FUNCTION_BLOCK FB_CylinderNexaHmi EXTENDS FB_Cylinder
VAR
	(* Hmi *)       			
	_Hmi						: TcNexa_Devices_TcDeviceBase.FB_DeviceNexaHmi(deviceType:= 'cylinders');
	_onHmiConnection			: Tc2_Standard.R_TRIG;
	_isHmiConnected				: BOOL;
	_commandNameHP				: STRING;
	_commandNameWP				: STRING;
	_manualMode					: BOOL;
	_onResponseError			: Tc2_Standard.R_TRIG;
	_onResponsePass				: Tc2_Standard.R_TRIG;
	_interlockHPforOtherDevices	: STRING;
	_interlockWPforOtherDevices	: STRING;
	(* Control VAR *)
	_lastNotUsedSensorHP		: BOOL;
	_lastSensorHP				: BOOL;
	_lastNotUsedSensorWP		: BOOL;
	_lastSensorWP				: BOOL;
	_message					: STRING(255);
	_lastMessage				: STRING(255);
	(* Buttons *)
	_ButtonHP					: TcNexa_Devices_TcDeviceBase.FB_DeviceButtonNexaHmi(
									Hmi			:= _Hmi, 
									topic		:= 'general/buttons/HP/');
	_ButtonWP					: TcNexa_Devices_TcDeviceBase.FB_DeviceButtonNexaHmi(
									Hmi			:= _Hmi, 
									topic		:= 'general/buttons/WP/');
	(* Commands *)
	_requestHP					: BOOL;
	_requestWP					: BOOL;
END_VAR

METHOD PROTECTED _handleButtons
VAR_INPUT
END_VAR
(*----------------------------------------------------------------------------------------------*)
_ButtonHP.enabled:= NOT _interlockHP AND _manualMode;
_ButtonHP.focused:= valveHP;
_ButtonHP.name:= _commandNameHP;
_ButtonHP.FB_main();
(*----------------------------------------------------------------------------------------------*)
_ButtonWP.enabled:= NOT _interlockWP AND _manualMode;
_ButtonWP.focused:= valveWP;
_ButtonWP.name:= _commandNameWP;
_ButtonWP.FB_main();
(*----------------------------------------------------------------------------------------------*)
IF NOT _manualMode THEN RETURN; END_IF
IF _ButtonHP.onTap THEN	_requestHP:= TRUE; END_IF
IF _ButtonWP.onTap THEN	_requestWP:= TRUE; END_IF
(*----------------------------------------------------------------------------------------------*)
END_METHOD

METHOD PROTECTED _handleManual
VAR_INPUT
END_VAR
IF NOT _manualMode THEN
	_requestHP:= FALSE;
	_requestWP:= FALSE;
	_message:= 'Movement blocked: Not in manual mode';
ELSIF _interlockHP AND NOT _inHP THEN
	_message:= Tc2_Standard.CONCAT(STR1:= _commandNameHP, ' blocked: ');
	_message:= Tc2_Standard.CONCAT(STR1:= _message, _interlockMessageHP);
ELSIF _interlockWP AND NOT _inWP THEN
	_message:= Tc2_Standard.CONCAT(STR1:= _commandNameWP, ' blocked: ');
	_message:= Tc2_Standard.CONCAT(STR1:= _message, _interlockMessageWP);
ELSE
	_message:= '';
	(* HP *)
	IF _requestHP THEN
		moveToHP(Response:= _InternalResponse);
		_requestHP:= FALSE;
	END_IF
	(* HP *)
	IF _requestWP THEN
		moveToWP(Response:= _InternalResponse);
		_requestWP:= FALSE;
	END_IF
END_IF
END_METHOD

METHOD PROTECTED _onConnection
VAR_INPUT
END_VAR
IF NOT _onHmiConnection.Q THEN RETURN; END_IF

(* Publish *)
_Hmi.publish(
	topic	:= 'general/sensorTagHP',
	payload	:= _sensorTagHP);
_Hmi.publish(
	topic	:= 'general/sensorTagWP',
	payload	:= _sensorTagWP);
END_METHOD

METHOD PROTECTED _publishTopics
VAR_INPUT
END_VAR
IF NOT _isHmiConnected THEN RETURN; END_IF
(*----------------------------------------------------------------------------------------------*)
IF (_lastNotUsedSensorHP <> _notUsedSensorHP) OR _onHmiConnection.Q THEN
	_lastNotUsedSensorHP:= _notUsedSensorHP;
	_Hmi.publish(
		topic	:= 'general/notUsedSensorHP',
		payload	:= BOOL_TO_STRING(_notUsedSensorHP));
END_IF
(*----------------------------------------------------------------------------------------------*)
IF (_lastSensorHP <> sensorHP) OR _onHmiConnection.Q THEN
	_lastSensorHP:= sensorHP;
	_Hmi.publish(
		topic	:= 'general/sensorHP',
		payload	:= BOOL_TO_STRING(sensorHP));
END_IF
(*----------------------------------------------------------------------------------------------*)
IF (_lastNotUsedSensorWP <> _notUsedSensorWP) OR _onHmiConnection.Q THEN
	_lastNotUsedSensorWP:= _notUsedSensorWP;
	_Hmi.publish(
		topic	:= 'general/notUsedSensorWP',
		payload	:= BOOL_TO_STRING(_notUsedSensorWP));
END_IF
(*----------------------------------------------------------------------------------------------*)
IF (_lastSensorWP <> sensorWP) OR _onHmiConnection.Q THEN
	_lastSensorWP:= sensorWP;
	_Hmi.publish(
		topic	:= 'general/sensorWP',
		payload	:= BOOL_TO_STRING(sensorWP));
END_IF
(*----------------------------------------------------------------------------------------------*)
IF (_message <> _lastMessage) OR _onHmiConnection.Q THEN
	_lastMessage:= _message;
	_Hmi.publish(
		topic	:= 'general/message',
		payload	:= _message);
END_IF
(*----------------------------------------------------------------------------------------------*)
END_METHOD

METHOD FB_init : BOOL
VAR_INPUT
	bInitRetains 	: BOOL; // if TRUE, the retain variables are initialized (warm start / cold start)
	bInCopyCode 	: BOOL;  // if TRUE, the instance afterwards gets moved into the copy code (online change)
	name			: STRING;
	tag				: STRING;
	sensorTagHP		: STRING;
	sensorTagWP		: STRING;
	commandNameHP	: STRING;
	commandNameWP	: STRING;
	cellTag			: STRING;
	stationTag		: STRING;
END_VAR
THIS^._commandNameHP:= commandNameHP;
THIS^._commandNameWP:= commandNameWP;

THIS^._Hmi.cellTag:= cellTag;
THIS^._Hmi.stationTag:= stationTag;
THIS^._Hmi.deviceTag:= tag;
THIS^._Hmi.deviceName:= name;

_interlockHPforOtherDevices:= Tc2_Standard.CONCAT(STR1:= _nameTag, STR2:= ' not in ');
_interlockHPforOtherDevices:= Tc2_Standard.CONCAT(STR1:= _interlockHPforOtherDevices, STR2:= _commandNameHP);
_interlockHPforOtherDevices:= Tc2_Standard.CONCAT(STR1:= _interlockHPforOtherDevices, STR2:= ' position');
_interlockWPforOtherDevices:= Tc2_Standard.CONCAT(STR1:= _nameTag, STR2:= ' not in ');
_interlockWPforOtherDevices:= Tc2_Standard.CONCAT(STR1:= _interlockWPforOtherDevices, STR2:= _commandNameWP);
_interlockWPforOtherDevices:= Tc2_Standard.CONCAT(STR1:= _interlockWPforOtherDevices, STR2:= ' position');
END_METHOD

METHOD PUBLIC FB_main
VAR_INPUT
END_VAR
SUPER^.FB_main();
_Hmi.FB_main();
_isHmiConnected:= _Hmi.isConnected;
_onHmiConnection(CLK:= _isHmiConnected);

_onConnection();
_publishTopics();
_handleButtons();
_handleManual();
END_METHOD

PROPERTY PUBLIC hostName : Tc2_System.T_MaxString
GET
hostName:= _Hmi.hostName;
END_GET
SET
_Hmi.hostName:= hostName;
END_SET
END_PROPERTY

PROPERTY PUBLIC hostPort : UINT
GET
hostPort:= _Hmi.hostPort;
END_GET
SET
_Hmi.hostPort:= hostPort;
END_SET
END_PROPERTY

PROPERTY interlockMessageHP : STRING(255)
GET
interlockMessageHP:= _interlockHPforOtherDevices;
END_GET
END_PROPERTY

PROPERTY interlockMessageWP : STRING(255)
GET
interlockMessageWP:= _interlockWPforOtherDevices;
END_GET
END_PROPERTY

PROPERTY manualMode : BOOL
GET
manualMode:= _manualMode;
END_GET
SET
_manualMode:= manualMode;
END_SET
END_PROPERTY

END_FUNCTION_BLOCK

(* stored: Version 1.1.0.1, ProductVersion 3.1.4026.17
   POU FB_CylinderNexaHmi: Id {a06e4a05-335d-41d8-bd6c-a9681a788555}, SpecialFunc None
   Folder Property: Id {02bde9a1-f084-0783-1fff-3b723a4f65ea}
   Folder Protected: Id {6f4f0496-5df3-4fdf-84ef-53779d8cadea}
   Method _handleButtons: Id {97794b87-e193-0072-13ea-f292d2ee2590}
   Method _handleManual: Id {7761fac9-f156-0d0e-1a07-34609e03ce5e}
   Method _onConnection: Id {66b7bbd5-26b9-4e3b-9129-d1227eacf7a1}
   Method _publishTopics: Id {f423ba49-c089-4fda-9965-66ea711d1b7c}
   Method FB_init: Id {89db22b4-7f64-0e0e-2f77-f5ba4ba17cbf}
   Method FB_main: Id {7288df59-cdb5-4cea-a1e3-32fbb9d17051}
   Property hostName: Id {7e5636fe-132a-0acc-1ae3-2ce97c5d5e86}
   Get Get: Id {7ba73824-d409-008c-05f0-177e106229c1}
   Set Set: Id {5bc415cc-d214-0cda-1aae-cee1fbf8fc6f}
   Property hostPort: Id {14cbd58c-5849-0244-3c79-cc8263901a1f}
   Get Get: Id {7d30d306-3ede-0146-0783-d5b9c74d5ee9}
   Set Set: Id {fed14df9-ad74-08c3-2cc2-5702d4cb36cf}
   Property interlockMessageHP: Id {38f74a37-690f-0b2c-3988-cd0be520935e}
   Get Get: Id {2ab42182-b181-0ed9-3c98-ac94fe5e55c6}
   Property interlockMessageWP: Id {73b1be68-b97c-03d8-2c32-42db0d213a42}
   Get Get: Id {99159a4b-3f50-0de6-03a9-e9eecf9304ad}
   Property manualMode: Id {302ce693-5704-0317-16e6-0b6e70ea6c09}
   Get Get: Id {1598543b-157f-0471-2ca8-d160363d5541}
   Set Set: Id {b370ce93-280e-0394-1067-40a0982f23ac} *)
